PROGRAM MAIN
VAR
	Axis			:	AXIS_REF;

	fbPower			:	MC_Power;
	bEnable			:	BOOL;
	bIsAxisReady	:	BOOL;
	
	fbMoveAbsolute	:	MC_MoveAbsolute;
	bExecute		:	BOOL;
	fPosition		:	LREAL;
	fVelocity		:	LREAL;
	bBusy			:	BOOL;
	bDone			:	bool;
END_VAR

Axis(); // Axis 정보 갱신

fbPower(
	Axis := Axis,
	Enable := bEnable,
	Enable_Positive := bEnable,
	Enable_Negative := bEnable,
	Status => bIsAxisReady // Axis가 동작할 준비가 왼료되면 TRUE
);

fbMoveAbsolute(
	Axis := Axis,
	Execute := bExecute,
	Position := fPosition,
	Velocity := fVelocity,
	Busy => bBusy,
	Done => bDone 
);

END_PROGRAM

(* stored: Version 1.1.0.1, ProductVersion 3.1.4024.5
   POU MAIN: Id {f064d8f9-778d-4913-a948-2610455ff419}, SpecialFunc None *)
